PROGRAM IP236
VAR
	timer				: TON;
	nState				: INT := STATE_INIT;
	
	fbInit236_01_5500			: FB_InitPM;
	fbInit236_02_5500			: FB_InitPM;
	fbInit236_03_5500			: FB_InitPM;
	fbInit236_04_5500			: FB_InitPM;
	fbInit236_05_5500			: FB_InitPM;
	fbInit236_06_5500			: FB_InitPM;
	fbInit236_07_5500			: FB_InitPM;
	fbInit236_08_5500			: FB_InitPM;
	fbInit236_11_5500			: FB_InitPM;
	fbInit236_33_5500			: FB_InitPM;
	fbInit236_38_5500			: FB_InitPM;
	
	fbRead236_01_5500			: FB_ReadPM5500;
	fbRead236_02_5500			: FB_PM_ION_9000;
	
	//Update 29-08-2022
	fbRead236_03_5500			: FB_ReadPM5350;
	
	fbRead236_04_5500			: FB_PM_ION_9000;
	
	//Update 29-08-2022
	fbRead236_05_5500			: FB_ReadPM5350;
	//Update 29-08-2022
	fbRead236_06_5500			: FB_ReadPM5350;
	
	
	fbRead236_07_5500			: FB_ReadPM5500;
	fbRead236_08_5500			: FB_ReadPM5500;
	fbRead236_11_5500			: FB_ReadPM5500;
	fbRead236_33_5500			: FB_ReadPM5500;
	fbRead236_38_5500			: FB_ReadPM5500;
	
	nCount						: DINT;
END_VAR

VAR CONSTANT
	STATE_INIT			:	INT		:= 0;
	STATE_WAIT_CMD		: 	INT		:= 5;
	STATE_READ1			:	INT		:= 10;
	STATE_READ2			:	INT		:= 20;
	STATE_READ3			:	INT		:= 30;
	STATE_READ4			:	INT		:= 40;
	STATE_READ5			:	INT		:= 50;
	STATE_READ6			:	INT		:= 60;
	STATE_READ7			:	INT		:= 70;
	STATE_READ8			:	INT		:= 80;
	STATE_READ11		:	INT		:= 110;
	STATE_READ33		:	INT		:= 330;
	STATE_READ38		:	INT		:= 380;
END_VAR

CASE nState OF
	STATE_INIT:
		fbInit236_01_5500(	sIpAddress	:= '10.91.37.236',
							nPort		:= 502,
							nUnitID		:= 1,
							PM			:= pmDev.DB06_01_5500);
		fbInit236_02_5500(	sIpAddress	:= '10.91.37.230',
							nPort		:= 502,
							nUnitID		:= 255,
							PM			:= pmDev.DB06_02_5500);
		fbInit236_03_5500(	sIpAddress	:= '10.91.37.236',
							nPort		:= 502,
							nUnitID		:= 3,
							PM			:= pmDev.DB06_03_5500);
		fbInit236_04_5500(	sIpAddress	:= '10.91.37.229',
							nPort		:= 502,
							nUnitID		:= 255,
							PM			:= pmDev.DB06_04_5500);
		fbInit236_05_5500(	sIpAddress	:= '10.91.37.236',
							nPort		:= 502,
							nUnitID		:= 5,
							PM			:= pmDev.DB06_05_5500);
							
		fbInit236_06_5500(	sIpAddress	:= '10.91.37.236',
							nPort		:= 502,
							nUnitID		:= 6,
							PM			:= pmDev.DB06_06_5500);
							
		fbInit236_07_5500(	sIpAddress	:= '10.91.37.236',
							nPort		:= 502,
							nUnitID		:= 7,
							PM			:= pmDev.DB06_07_5500);
							
		fbInit236_08_5500(	sIpAddress	:= '10.91.37.236',
							nPort		:= 502,
							nUnitID		:= 8,
							PM			:= pmDev.DB06_08_5500);
							
		fbInit236_11_5500(	sIpAddress	:= '10.91.37.236',
							nPort		:= 502,
							nUnitID		:= 11,
							PM			:= pmDev.DB06_11_5500);
							
		fbInit236_33_5500(	sIpAddress	:= '10.91.37.236',
							nPort		:= 502,
							nUnitID		:= 33,
							PM			:= pmDev.DB06_33_5500);
							
		fbInit236_38_5500(	sIpAddress	:= '10.91.37.236',
							nPort		:= 502,
							nUnitID		:= 38,
							PM			:= pmDev.DB06_38_5500);
		
		timer(In:=TRUE, PT:= TIME_INIT);
		IF timer.Q THEN
			timer(In := FALSE);
			nState	:= STATE_WAIT_CMD;
		END_IF
		
	STATE_WAIT_CMD:
		;
		
	STATE_READ1:
		fbRead236_01_5500(
			bExecute:=TRUE,
			PM:= pmDev.DB06_01_5500);
		IF NOT fbRead236_01_5500.Q THEN
			nState	:= STATE_READ2;
			fbRead236_01_5500(
				bExecute:=FALSE,
				PM:= pmDev.DB06_01_5500);
		END_IF
		
	STATE_READ2:
		fbRead236_02_5500(
			bExecute:=TRUE,
			PM:= pmDev.DB06_02_5500);
		IF NOT fbRead236_02_5500.Q THEN
			nState	:= STATE_READ3;
			fbRead236_02_5500(
				bExecute:=FALSE,
				PM:= pmDev.DB06_02_5500);
		END_IF	
	
	STATE_READ3:
	
		fbRead236_03_5500(
			bExecute:=TRUE,
			PM:= pmDev.DB06_03_5500);
		IF NOT fbRead236_03_5500.Q THEN
			nState	:= STATE_READ4;
			fbRead236_03_5500(
				bExecute:=FALSE,
				PM:= pmDev.DB06_03_5500);
		END_IF	
		
	STATE_READ4:
		fbRead236_04_5500(
			bExecute:=TRUE,
			PM:= pmDev.DB06_04_5500);
		IF NOT fbRead236_04_5500.Q THEN
			nState	:= STATE_READ5;
			fbRead236_04_5500(
				bExecute:=FALSE,
				PM:= pmDev.DB06_04_5500);
		END_IF	
		
	STATE_READ5:
	
		fbRead236_05_5500(
			bExecute:=TRUE,
			PM:= pmDev.DB06_05_5500);
		IF NOT fbRead236_05_5500.Q THEN
			nState	:= STATE_READ6;
			fbRead236_05_5500(
				bExecute:=FALSE,
				PM:= pmDev.DB06_06_5500);
		END_IF	
		
	STATE_READ6:
	
		
		fbRead236_06_5500(
			bExecute:=TRUE,
			PM:= pmDev.DB06_06_5500);
		IF NOT fbRead236_06_5500.Q THEN
			nState	:= STATE_READ7;
			fbRead236_06_5500(
				bExecute:=FALSE,
				PM:= pmDev.DB06_06_5500);
		END_IF	
		
	STATE_READ7:
		fbRead236_07_5500(
			bExecute:=TRUE,
			PM:= pmDev.DB06_07_5500);
		IF NOT fbRead236_07_5500.Q THEN
			nState	:= STATE_READ8;
			fbRead236_07_5500(
				bExecute:=FALSE,
				PM:= pmDev.DB06_07_5500);
		END_IF
		
	STATE_READ8:
		fbRead236_08_5500(
			bExecute:=TRUE,
			PM:= pmDev.DB06_08_5500);
		IF NOT fbRead236_08_5500.Q THEN
			nState	:= STATE_READ11;
			fbRead236_08_5500(
				bExecute:=FALSE,
				PM:= pmDev.DB06_08_5500);
		END_IF
		
	STATE_READ11:
		fbRead236_11_5500(
			bExecute:=TRUE,
			PM:= pmDev.DB06_11_5500);
		IF NOT fbRead236_11_5500.Q THEN
			nState	:= STATE_READ33;
			fbRead236_11_5500(
				bExecute:=FALSE,
				PM:= pmDev.DB06_11_5500);
		END_IF
		
	STATE_READ33:
		fbRead236_33_5500(
			bExecute:=TRUE,
			PM:= pmDev.DB06_33_5500);
		IF NOT fbRead236_33_5500.Q THEN
			nState	:= STATE_READ38;
			fbRead236_33_5500(
				bExecute:=FALSE,
				PM:= pmDev.DB06_33_5500);
		END_IF
		
	STATE_READ38:
		fbRead236_38_5500(
			bExecute:=TRUE,
			PM:= pmDev.DB06_38_5500);
		IF NOT fbRead236_38_5500.Q THEN
			nState	:= STATE_WAIT_CMD;
			fbRead236_38_5500(
				bExecute:=FALSE,
				PM:= pmDev.DB06_38_5500);
		END_IF
		
END_CASE

PROPERTY Busy : Bool
GET
Busy := nState <> STATE_WAIT_CMD;
END_GET
END_PROPERTY

METHOD Mr_Read : BOOL
VAR_INPUT
END_VAR
IF nState = STATE_WAIT_CMD THEN
	nState := STATE_READ1;
END_IF
END_METHOD

END_PROGRAM

(* stored: Version 1.1.0.1, ProductVersion 3.1.4024.12
   POU IP236: Id {acd8d4c0-f512-44fa-adf7-17da8b59fda0}, SpecialFunc None
   Property Busy: Id {53280eb6-6933-4f72-be91-b659b9f4b362}
   Get Get: Id {f04f0807-29d0-4fd1-98f0-6dbddec742e2}
   Method Mr_Read: Id {3ea01a05-f97a-4bc6-8625-cb244e954181} *)
